FUNCTION_BLOCK FB_BottleFiller
VAR_INPUT
	bisTankEmpty : BOOL;
	bLevelSensor : BOOL;
END_VAR
VAR
	bFillingValve : BOOL;
	bValvePressure : DINT ;
	
END_VAR
VAR_OUTPUT
	bFilling : BOOL;
	bSpeed : DINT;
END_VAR

METHOD SetValvePressure
VAR_INPUT
	bPressureValue : DINT;
END_VAR
bValvePressure := bPressureValue;
bSpeed := bValvePressure -10;
END_METHOD

METHOD StartFilling : BOOL
VAR_INPUT
END_VAR
IF bisTankEmpty THEN
	bFilling := bFillingValve := TRUE;
END_IF
END_METHOD

METHOD StopFilling : BOOL
VAR_INPUT
END_VAR
IF bLevelSensor THEN
	bFilling := bFillingValve := FALSE;
END_IF
END_METHOD

END_FUNCTION_BLOCK

(* stored: Version 1.1.0.1, ProductVersion 3.1.4024.16
   POU FB_BottleFiller: Id {9cb8cf01-0ea3-43ab-b787-0cb5775d9ae4}, SpecialFunc None
   Method SetValvePressure: Id {f3c5295d-588f-4712-9439-4d32f5671a47}
   Method StartFilling: Id {851d32b8-1dd9-4740-bfa9-12e36ba93498}
   Method StopFilling: Id {feb6e664-1480-4b85-8cdd-d94997f7425d} *)
